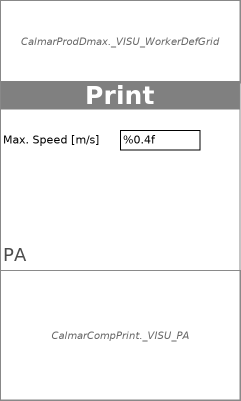
VISUALIZATION _VISU_WorkerWeu_Print  // 241x401
VAR_IN_OUT
  m_Inst : FB_WorkerDefGrid_Print_WEU;
END_VAR
    Frame (0,0 241x83)
        shows CalmarProdDmax._VISU_WorkerDefGrid(m_Inst := m_Inst)
    Label (0,240 240x30), "PA"
    Rectangle (0,80 240x30), "Print"
    Frame (0,270 241x131)
        shows CalmarCompPrint._VISU_PA(m_Inst := m_Inst.fbPa)
    Rectangle (0,130 120x20), "Max. Speed [m/s]"
    Rectangle (120,130 80x20), "%0.4f", text variable: m_Inst.fMaxSpeed
END_VISUALIZATION

(* stored: Version 1.1.0.1, ProductVersion 3.1.4024.11
   Visu _VISU_WorkerWeu_Print: Id {106bf08b-3246-4506-8c48-e81ae7b17b40} *)
